PROGRAM INTERNAL PRG_TESTS

(* Instantiate test suites here. Naming convention for tests should be a suffix with _Tests.
Good practice for creating test methods is to end them with _test as well. *)
VAR
	FlowControllerTests	: FB_FlowController_Tests;
	FlowUnitTests		: FB_FlowUnits_Tests;
	GasTypesTests		: FB_GasTypes_Tests;
END_VAR

// Run tests in paralel
//TcUnit.RUN();

// Run tests in sequence, one after the other. Uncomment if required.
TcUnit.RUN_IN_SEQUENCE();

END_PROGRAM

(* stored: Version 1.1.0.1, ProductVersion 3.1.4024.16
   POU PRG_TESTS: Id {8a697354-56fc-44b0-afc4-e6c08f5bd900}, SpecialFunc None *)
